Staubli VAL3: ros_server.pjx

--- ros_server.pjx ---
Parameters version=s7.11 stackSize=5000 millimeterUnit=true
Program file=dataReceiver.pgx
Program file=dataStreamer.pgx
Program file=decodeMsgBody.pgx
Program file=decodeMsgHeader.pgx
Program file=decTrajPt.pgx
Program file=decTrajPtFull.pgx
Program file=encodeAck.pgx
Program file=encodeJState.pgx
Program file=encodeStatus.pgx
Program file=encPrefixHeader.pgx
Program file=encTrajPtAck.pgx
Program file=encTrajPtFAck.pgx
Program file=fetchStatus.pgx
Program file=initParams.pgx
Program file=interpolateVel.pgx
Program file=motionControl.pgx
Program file=pushMotion.pgx
Program file=recvData.pgx
Program file=recvHeartbeat.pgx
Program file=recvMsgBody.pgx
Program file=recvMsgHeader.pgx
Program file=recvTrajPt.pgx
Program file=recvTrajPtFull.pgx
Program file=screenUpdate.pgx
Program file=sendAck.pgx
Program file=sendData.pgx
Program file=sendRosMsg.pgx
Program file=setupRosMsgs.pgx
Program file=start.pgx
Program file=stop.pgx
Program file=toJointArrayRad.pgx
Program file=toJointRxDeg.pgx
Data file=ros_server.dtx
Library alias=libQueueFuncs path=../ros_libs/QueueFuncs/QueueFuncs.pjx
Library alias=libInterface path=../ros_libs/UserInterface/interfaceDefault/interfaceDefault.pjx autoload=false
Type name=RosSimpleMsg path=../ros_libs/RosSimpleMsg/RosSimpleMsg.pjx
Type name=RobotStatusMsg path=../ros_libs/RobotStatusMsg/RobotStatusMsg.pjx
Type name=JointStateMsg path=../ros_libs/JointStateMsg/JointStateMsg.pjx
Type name=JointTrajPtMsg path=../ros_libs/JointTrajPtMsg/JointTrajPtMsg.pjx
Type name=JointTrajPtFMsg path=../ros_libs/JointTrajPtFMsg/JointTrajPtFMsg.pjx
Type name=JointFbkMsg path=../ros_libs/JointFbkMsg/JointFbkMsg.pjx
Type name=MotionCmd path=../ros_libs/MotionCmd/MotionCmd.pjx
Type name=Header path=../ros_libs/Header/Header.pjx
Type name=Prefix path=../ros_libs/Prefix/Prefix.pjx
Type name=Body path=../ros_libs/Body/Body.pjx
Type name=Queue path=../ros_libs/Queue/Queue.pjx

--- start.pgx ---
program start()
  local num l_nFbkPeriod
  local num l_nMotionPeriod
  local num l_nTrajPeriod
  local num l_nScreenUpdate
  local string l_sVersionMajor
  local num l_nVersionMajor
  local bool l_bOkMajor
  local string l_sVersionMinor
  local num l_nVersionMinor
  local bool l_bOkMinor
begin
  // Copyright (c) 2016, Ocado Technology - Robotics Research Team
  //
  // Licensed under the Apache License, Version 2.0 (the "License");
  // you may not use this file except in compliance with the License.
  // You may obtain a copy of the License at
  //
  //     http://www.apache.org/licenses/LICENSE-2.0
  //
  // Unless required by applicable law or agreed to in writing, software
  // distributed under the License is distributed on an "AS IS" BASIS,
  // WITHOUT WARRANTIES OR CONDITIONS OF ANY KIND, either express or implied.
  // See the License for the specific language governing permissions and
  // limitations under the License.


  // Load interface library for CS8 or CS9
  //
  // CS9 handles the UI differently than CS8, requires
  // the UI funtions to be loaded in seperate libraries

  if(mid(getVersion("System"),1,1) == "7")
    // CS8 - VAL 3 rev 7
    // Check for VAL 3 version >= 7.7
    l_sVersionMajor = mid(getVersion("VAL3"),1,1)
    l_sVersionMinor = mid(getVersion("VAL3"),2,1)
    toNum(l_sVersionMajor, l_nVersionMajor, l_bOkMajor)
    toNum(l_sVersionMinor, l_nVersionMinor, l_bOkMinor)
    if(!l_bOkMajor or !l_bOkMinor)
      popUpMsg("Error reading VAL 3 version")
      taskKill("ros_server~")
    endIf
    if( !((l_nVersionMajor == 7) and (l_nVersionMinor >= 7)))
      // VAL 3 version is too old
      popUpMsg("Error: VAL 3 version is < 7.7, socket communication will not work!")
      taskKill("ros_server~")
    endIf
    libInterface:libLoad("../ros_libs/UserInterface/interfaceCS8")
  elseIf(mid(getVersion("System"),1,1) == "8")
    // CS9 - VAL 3 rev 8
    libInterface:libLoad("../ros_libs/UserInterface/interfaceCS9")
  endIf

  // feedback task will run every 20ms (50Hz)
  l_nFbkPeriod=0.02
  //l_nFbkPeriod = 0.032 // 30Hz
  //l_nFbkPeriod = 0.05  // 20Hz
  //l_nFbkPeriod = 1.0   //  1Hz

  // motion control task will run every 4ms (250Hz)
  l_nMotionPeriod = 0.004
  //l_nMotionPeriod=0.012  // 83Hz
  //l_nMotionPeriod = 0.05 // 20Hz

  // data (trajectory) reception task will run every 4ms (250Hz)
  l_nTrajPeriod = 0.004
  // not in use at the moment
  l_nScreenUpdate = 1.0

  sStreamTaskName = "streamerTask"
  sTrajPtTaskName = "trajPtTask"
  sMotionTaskName = "motionTask"
  sScreenTaskName = "screenTask"
  sHtbtTaskName = "htbtTask"

  // initialise TCP/IP parameters
  call initParams()
  // setup prefix and header of ROS messages
  call setupRosMsgs()

  // socket connection status flags: initially disconnected
  nInConnFlag = 0
  nOutConnFlag = 0

  // flag defining whether velocity to be overwritten to max. vel.
  bOverwriteVel = false

  nPtsPopped = 0
  nMovePts = 0

  // flush buffer of incoming socket
  clearBuffer(siTcpIpMotion)
  // flush buffer of outgoing socket
  clearBuffer(siTcpIpFbk)

  // check if robot is not in emergency stop and wait until estop is reset
  if(esStatus() == 2)
    popUpMsg("Please reset E-Stop")
    wait(esStatus() < 2)
  endIf

  // before anything else, enable power (only works if robot is in remote mode)
  if(!isPowered())
    if(workingMode() >= 4)
      do
        enablePower()
        delay(2)
      until isPowered()
    else
      popUpMsg("Power must be enabled manually")
    endIf
  endIf

  // reset motion, potentially setting a start joint position for calling autoConnect() in the future
  resetMotion()

  // create joint state and robot status streamer task to send data to industrial_robot_client
  taskCreateSync sStreamTaskName, l_nFbkPeriod, bFbkOverrun, dataStreamer()

  // create trajectory point task to receive data from industrial_robot_client
  taskCreateSync sTrajPtTaskName, l_nTrajPeriod, bTrajPtOverrun, dataReceiver()
  //taskCreate sTrajPtTaskName, 100, dataReceiver()

  // create motion task to synchronously apply motion commands to robot
  taskCreateSync sMotionTaskName, l_nMotionPeriod, bMotionOverrun, motionControl()

  // create synchronous task to update screen
  //taskCreateSync sScreenTaskName, l_nScreenUpdate, bScreenOverrun, screenUpdate()
  taskCreate sScreenTaskName, 10, screenUpdate()

  // create asynchronous task to receive heartbeat on port 11002
  taskCreate sHtbtTaskName, 10, recvHeartbeat()

end

--- motionControl.pgx ---
public program motionControl()
  local MotionCmd l_mTrajPt
  local bool l_bFlag
  local MotionCmd l_motion
  local num l_nElems
  local bool bLastPt
  local num nPrevVel
begin
  // Copyright (c) 2016, Ocado Technology - Robotics Research Team
  //
  // Licensed under the Apache License, Version 2.0 (the "License");
  // you may not use this file except in compliance with the License.
  // You may obtain a copy of the License at
  //
  //     http://www.apache.org/licenses/LICENSE-2.0
  //
  // Unless required by applicable law or agreed to in writing, software
  // distributed under the License is distributed on an "AS IS" BASIS,
  // WITHOUT WARRANTIES OR CONDITIONS OF ANY KIND, either express or implied.
  // See the License for the specific language governing permissions and
  // limitations under the License.



  nMoveId = -1

  while(true)
    // check connection status, and whether to stop motion
    if(nInConnFlag == 1 and nOutConnFlag == 1 and bStopNow == false)

      // process trajectory point from trajectory buffer
      call libQueueFuncs:getNumElems(qTrajPtBuffer, l_nElems)
      if(l_nElems > 0)
        call libQueueFuncs:pop(qTrajPtBuffer,l_mTrajPt, l_bFlag)
        if(l_bFlag == true)
          nPtsPopped = nPtsPopped + 1
          call libQueueFuncs:push(qMoveBuffer,l_mTrajPt,l_bFlag)
        endIf
      endIf

      // process motion command from move buffer
      // @TODO move buffer should have elements previously interpolated to ensure they are 4 ms apart
      call libQueueFuncs:getNumElems(qMoveBuffer, l_nElems)
      if(l_nElems > 0)
        call libQueueFuncs:pop(qMoveBuffer,l_motion,l_bFlag)
        if(l_bFlag == true)
          nMovePts = nMovePts + 1

          // Velocity buffer to smooth out last traj point
          nVel[1] = nVel[0]
          nVel[0] = rosTrajPtMsg.jointTrajPt.nVelocity

          // contrary to what we did earlier, we unconditionally add the traj pt to the motion queue:
          // there doesn't appear to be a way to compare the 'current pose' of the robot to the pts
          // in the trajectory at the appropriate time (ie: when the robot is in motion and about to
          // start executing the segment towards 'l_motion').
          // Checking for dist(l_motion, herej()) (pseudo code) would not be correct as there will
          // always be a delay in the data coming out of herej() and the actual pose of the robot.
          // @TODO potentially set move id according to sequence value

          // to detect the last point, its velocity is set to 2 (resulting in 200 here) before sending it. The previous pts velocity is used.
          if ((l_motion.mDesc.vel > 199.999) and (l_motion.nSequence != 0))
            bLastPt = true
            l_motion.mDesc.vel = nPrevVel
          else
            bLastPt = false
            nPrevVel = l_motion.mDesc.vel
          endIf


          l_motion.mDesc.blend=joint
          l_motion.mDesc.leave=0.5
          l_motion.mDesc.reach=0.5

          nMoveId = movej(l_motion.jJointRx, tTool, l_motion.mDesc)

          // do not use blending for last pt
          if (bLastPt)
            waitEndMove()
          endIf
        endIf
      endIf
    else
      // stop immediately -- resetMotion() also resets moveId
      resetMotion()
      // clear buffers
      call libQueueFuncs:clear(qTrajPtBuffer)
      call libQueueFuncs:clear(qMoveBuffer)
      bStopNow = false

      // debug
      nPtsPopped = 0
      nMovePts = 0
    endIf

    nMotionProgress = getMoveId()

    // sequence task
    delay(0)
  endWhile
end

--- pushMotion.pgx ---
public program pushMotion(num& x_nMsgRecvState)
  local bool l_bOk
  local num l_nCounter
  local num l_nJointError
  local MotionCmd l_mTrajPt
begin
  // Copyright (c) 2016, Ocado Technology - Robotics Research Team
  //
  // Licensed under the Apache License, Version 2.0 (the "License");
  // you may not use this file except in compliance with the License.
  // You may obtain a copy of the License at
  //
  //     http://www.apache.org/licenses/LICENSE-2.0
  //
  // Unless required by applicable law or agreed to in writing, software
  // distributed under the License is distributed on an "AS IS" BASIS,
  // WITHOUT WARRANTIES OR CONDITIONS OF ANY KIND, either express or implied.
  // See the License for the specific language governing permissions and
  // limitations under the License.



  switch rosGenericMsg.header.nMsgType
    case nStdMsgType["JOINT_TRAJ_PT"]
      l_mTrajPt.nSequence=rosTrajPtMsg.jointTrajPt.nSeq

      // ROS joint position values are in rad, but VAL3 uses degrees
      call toJointRxDeg(rosTrajPtMsg.jointTrajPt.nJoints, l_mTrajPt.jJointRx)

      // from industrial_robot_client/src/joint_trajectory_interface.cpp
      // JointTrajectoryInterface::trajectory_to_msgs()
      // JointTrajectoryInterface::calc_speed()
      // velocity is converted to a scalar value representing % of max velocity,
      // such that 0.2 = 20% of maximum joint speed
      if(rosTrajPtMsg.jointTrajPt.nVelocity > 1.99)
        l_mTrajPt.mDesc.vel = 200
      else
        l_mTrajPt.mDesc.vel= limit((rosTrajPtMsg.jointTrajPt.nVelocity * 100), 0, 100)
      endIf
      l_mTrajPt.nDuration=rosTrajPtMsg.jointTrajPt.nDuration

    break
    case nStdMsgType["JOINT_TRAJ_PT_FULL"]
      l_mTrajPt.nSequence=rosTrajPtFMsg.jointTrajPtFull.nSeq
      l_mTrajPt.nDuration=rosTrajPtFMsg.jointTrajPtFull.nTime

      // ROS joint position values are in rad, but VAL3 uses degrees
      call toJointRxDeg(rosTrajPtFMsg.jointTrajPtFull.nPositions, l_mTrajPt.jJointRx)

      // from industrial_robot_client/src/joint_trajectory_interface.cpp
      // JointTrajectoryInterface::trajectory_to_msgs()
      // JointTrajectoryInterface::calc_speed()
      // velocity is converted to a scalar value representing % of max velocity,
      // such that 0.2 = 20% of maximum joint speed
      l_mTrajPt.mDesc.vel= limit((rosTrajPtFMsg.jointTrajPtFull.nVelocities[0] * 100), 0, 100)
      // not sure about accelerations as yet
      l_mTrajPt.mDesc.accel=rosTrajPtFMsg.jointTrajPtFull.nAccelerations[0]
      l_mTrajPt.mDesc.decel=l_mTrajPt.mDesc.accel
    break
    default
    break
  endSwitch

  // see github.com/ros-industrial/industrial_core/simple_message/include/simple_message/joint_traj_pt.h
  if(l_mTrajPt.nSequence==-4)
    // set flag to stop immediately
    bStopNow=true
  else
    // check whether velocity value should be overwritten with value set on teach pendant
    if(bOverwriteVel == true)
      // overwrite velocity (and acceleration - ?)
      //l_mTrajPt.mDesc.vel = getMonitorSpeed()
      // explicitly setting accel and decel to VAL3 default values
      l_mTrajPt.mDesc.accel = mNomSpeed.accel
      l_mTrajPt.mDesc.decel = mNomSpeed.decel
    endIf
    // only push motion into buffer if not a STOP message
    // and if joint positions are within software joint limits
    // and if velocity is greater than zero (beucase movej() will not accept vel <= 0)
    if(isInRange(l_mTrajPt.jJointRx) and l_mTrajPt.mDesc.vel > 0)
      call libQueueFuncs:push(qTrajPtBuffer,l_mTrajPt,l_bOk)
    else
      l_bOk = false
    endIf

    if(l_bOk==false)
      // could not push trajectory point into buffer
      // thus ACK should flag FAILURE, but only if comm type is request
      if(rosGenericMsg.header.nCommType==nCommType["SERVICE_REQUEST"])
        switch rosGenericMsg.header.nMsgType
          case nStdMsgType["JOINT_TRAJ_PT"]
            rosTrajPtAck.header.nReplyCode=2
          break
          case nStdMsgType["JOINT_TRAJ_PT_FULL"]
            rosTrajPtFAck.header.nReplyCode=2
          break
          default
          break
        endSwitch
      endIf
    endIf
  endIf
  // check whether ACK should be sent
  if(rosGenericMsg.header.nCommType == nCommType["SERVICE_REQUEST"])
    // comm type request requires ACK
    x_nMsgRecvState = nAck
  else
    // other comm types (e.g., topic) does not require ACK, hence skip state
    x_nMsgRecvState = nReset
  endIf
end
